PROGRAM Teste
VAR

END_VAR

FOR i := 1 TO GVL_TimeSchBABR.cNumberOfEventSchedules DO
	timeScheduler[i](
		timeToActivate:= GVL_TimeSchBABR.aTimeToSchActivate[actualDate.wDayOfWeek,i], 
		timeToDeactivate:= GVL_TimeSchBABR.aTimeToSchDeactivate[actualDate.wDayOfWeek,i], 
		actualTime:= actualDate, 
		bTurnOffOutput:= bTurnOffOutput, 
		bErr=> bErr, 
		sErr=> sErr, 
		bOut=> GVL_TimeSchBABR.abOutScheduler[i]);
END_FOR

END_PROGRAM

(* stored: Version 1.1.0.1, ProductVersion 3.1.4020.6
   POU Teste: Id {38722a99-fb9b-4890-b31c-8913a076df2a}, SpecialFunc None *)
